// TIA Portal project "ConveyorBeltSystem" (V15)
// The purpose of project is to create a transport string system

(* hardware
DEVICE "S7-1200 station_1"  S7-1200 Station
   slot 0: "Rack_0"  S7-1200 Rack  Rack  V1.0
   slot 1: "PLC_1"  CPU 1214C DC/DC/DC  6ES7 214-1AG40-0XB0  V4.2
*)

// ===== PLC "PLC_1"  CPU 1214C DC/DC/DC =====

VAR_GLOBAL   // PLC tag table "Default tag table"
   "Takeoff_at_End3" AT %I0.5 : Bool;
   "Regulation" AT %I0.6 : Bool;   // ustawienie trybu pracy: szybki / wolny
   "Divisor" AT %M1.0 : Bool;   // przelacznik
   "Divisor_Memory" AT %M1.1 : Bool;   // pamiec przelacznika
   "Conveyor_Belt_1_Input" AT %I0.1 : Bool;   // wejscie na transporter #1
   "Conveyor_Belt_2_Input" AT %I0.2 : Bool;   // wejscie na transporter #2 / potwierdzenie odebrania paczki dla transportera #1
   "Conveyor_Belt_1_Output" AT %Q0.1 : Bool;   // wyjscie transporera #1 - sterowanie silnikiem
   "Conveyor_Belt_3_Input" AT %I0.3 : Bool;   // wejscie na transporter #3 / potwierdzenie odebrania paczki dla transportera #2
   "Conveyor_Belt_2_Output" AT %Q0.2 : Bool;   // wyjscie transporera #2 - sterowanie silnikiem
   "Conveyor_Belt_3_Confirm" AT %I0.4 : Bool;   // potwierdzenie odebrania paczki
   "Conveyor_Belt_3_Output" AT %Q0.3 : Bool;   // wyjscie transporera #3 - sterowanie silnikiem
   "Regulation_Edge" AT %M0.6 : Bool;   // zbocze regulacji trybow pracy
   "Conveyor_Belt_2_Status" AT %Q0.5 : Bool;   // sygnal wyjsciowy informujacy czy znajduje sie towar na koncu linii #2
   "Conveyor_Belt_3_Status" AT %Q0.6 : Bool;   // sygnal wyjsciowy informujacy czy znajduje sie towar na koncu linii #3
   "Conveyor_Belt_1_Status" AT %Q0.4 : Bool;   // sygnal wyjsciowy informujacy czy znajduje sie towar na koncu linii #1
   "Conveyor_Belt_1_Malfunction" AT %M500.0 : Bool;   // pamiec o wystapieniu awarii na transporterze #1
   "Conveyor_Belt_2_Malfunction" AT %M500.1 : Bool;   // pamiec o wystapieniu awarii na transporterze #2
   "Conveyor_Belt_3_Malfunction" AT %M500.2 : Bool;   // pamiec o wystapieniu awarii na transporterze #3
   "Tag_1" AT %M501.0 : Bool;
   "Tag_2" AT %M501.1 : Bool;
   "generator" AT %M30.0 : Bool;   // generator dla kanalow alarmowych
   "Conveyor_Belt_1_Alarm" AT %Q1.0 : Bool;   // wyjscie dla sygnalu awarii na transporterze #1
   "Conveyor_Belt_2_Alarm" AT %Q1.1 : Bool;   // wyjscie dla sygnalu awarii na transporterze #2
   "Conveyor_Belt_3_Alarm" AT %Q1.2 : Bool;   // wyjscie dla sygnalu awarii na transporterze #3
   "Emergency_Memory_1" AT %M500.3 : Bool;
   "Emergency_Memory_2" AT %M500.4 : Bool;
   "Emergency_Memory_3" AT %M500.5 : Bool;
   "Emergency_3_Confirm" AT %I1.2 : Bool;   // potwierdzenie awarii dla transportera #3
   "Emergency_2_Confirm" AT %I1.1 : Bool;   // potwierdzenie awarii dla transportera #2
   "Emergency_1_Confirm" AT %I1.0 : Bool;   // potwierdzenie awarii dla transportera #1
END_VAR

DATA_BLOCK "ConveyorBelt1_DB"   // DB1
{ S7_Optimized_Access := 'TRUE' }
VERSION : 0.1
// stored: InstanceOfName ConveyorBelt
"ConveyorBelt"
BEGIN
END_DATA_BLOCK

DATA_BLOCK "ConveyorBelt2_DB"   // DB2
{ S7_Optimized_Access := 'TRUE' }
VERSION : 0.1
// stored: InstanceOfName ConveyorBelt
"ConveyorBelt"
BEGIN
END_DATA_BLOCK

DATA_BLOCK "ConveyorBelt3_DB"   // DB3
{ S7_Optimized_Access := 'TRUE' }
VERSION : 0.1
// stored: InstanceOfName ConveyorBelt
"ConveyorBelt"
BEGIN
END_DATA_BLOCK

FUNCTION_BLOCK "ConveyorBelt"   // FB1, LAD
TITLE = Taśmociąg
{ S7_Optimized_Access := 'TRUE' }
VERSION : 0.1
// Blok funkcyjny odpowiedzialny za logikę pracy taśmociągu
   VAR_INPUT
      On_Line : Bool;   // podanie towaru na wejscie transportera
      Deliver_Confirm : Bool;   // potwierdzenie odbioru przez nastepna linie
      Malfunction_Confirm : Bool;   // potwierdzenie awarii przez operatora
   END_VAR
   VAR_OUTPUT
      Motor_Status : Bool;   // sygnal sterujacy silnikiem
      Malfunction : Bool;   // sygnal informujacy o awarii
      Output_Signal : Bool;   // sygnal informujacy, ze na koncu linii znajduje sie paczka
   END_VAR
   VAR
      Motor_Work : Bool;   // sygnal wyjsciowy informujacy o ladunku na koncu toru
      Blocked : Bool;   // sygnal ustawiajacy blokade transportera
      Photodiode_at_Start : Bool;   // status fotodiody umieszczonej na poczatku
      Counter_at_Start : Word;   // licznik towaru na wejsciu
      Photodiode_at_End : Bool;   // status fotodiody umieszczonej na koncu toru
      Counter_at_End : Word;   // licznik towaru na wyjsciu
      Work_Time : Time;   // czas pracy transportera
      IEC_Timer_0_Instance_2 : TP_TIME;
   END_VAR
   VAR RETAIN
      Package_Counter__Instance : CTUD_INT;
      Package_at_End_Counter_0_DB : CTU_INT;
   END_VAR
   VAR
      Photodiode_at_Start_Instance : "Photodiode";
      Photodiode_at_End_Instance : "Photodiode";
   END_VAR
   VAR RETAIN
      Counter_at_Start_Instance : CTU_INT;
   END_VAR
   VAR_TEMP
      Edge_Counter_at_Start_ : Bool;   // pamiec zbocza licznika na poczatku
      Edge_Counter_at_End : Bool;   // pamiec zbocza licznika na koncu
      Photodiode_End_Edge : Bool;   // pamiec zbocza fotodiody na koncu
      Photodiode_Start_Edge : Bool;   // pamiec zbocza fotodiody na poczatku
   END_VAR
   VAR_TEMP   // added for the SCL form of the ladder/FBD networks
      _w1 : Bool;
   END_VAR
BEGIN

REGION Network 1: Fotodioda 1: wykrycie towaru na początku
   // jesli nie ma blokady i fotodioda wykryje paczke ustaw jej sygnal
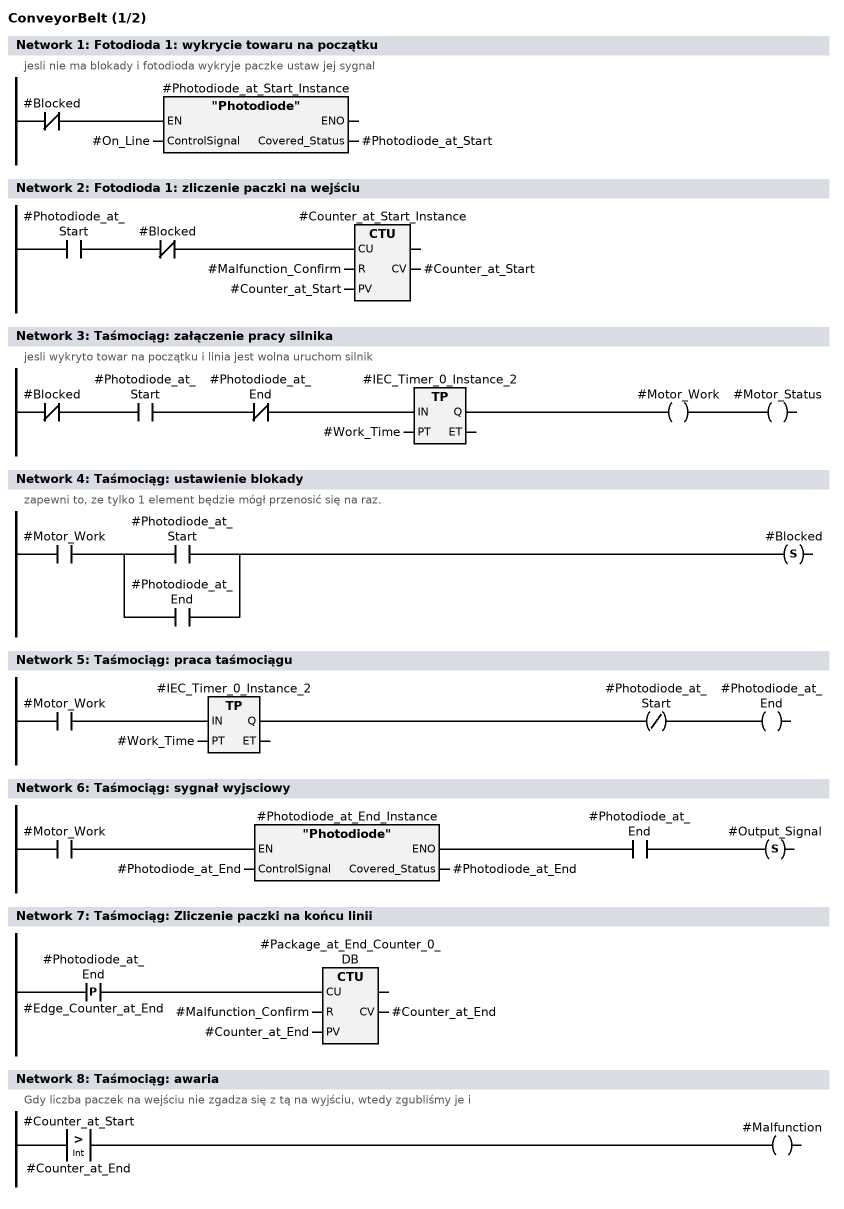
   RUNG wire#powerrail
      I_Contact( #Blocked )
      #Photodiode_at_Start_Instance(ControlSignal := #On_Line, Covered_Status => #Photodiode_at_Start)
   END_RUNG
   // the same network as SCL:
   IF NOT #Blocked THEN
       #Photodiode_at_Start_Instance(ControlSignal := #On_Line, Covered_Status => #Photodiode_at_Start);   // "Photodiode"
   END_IF;
END_REGION

REGION Network 2: Fotodioda 1: zliczenie paczki na wejściu
   #Counter_at_Start_Instance(CU := #Photodiode_at_Start AND NOT #Blocked,   // CTU
                           R := #Malfunction_Confirm,
                           PV := #Counter_at_Start,
                           CV => #Counter_at_Start);
END_REGION

REGION Network 3: Taśmociąg: załączenie pracy silnika
   // jesli wykryto towar na początku i linia jest wolna uruchom silnik
   #IEC_Timer_0_Instance_2(IN := NOT #Blocked AND #Photodiode_at_Start AND NOT #Photodiode_at_End,   // TP
                           PT := #Work_Time);
   #Motor_Work := #IEC_Timer_0_Instance_2.Q;
   #Motor_Status := #IEC_Timer_0_Instance_2.Q;
END_REGION

REGION Network 4: Taśmociąg: ustawienie blokady
   // zapewni to, ze tylko 1 element będzie mógł przenosić się na raz.
   RUNG wire#powerrail
      Contact( #Motor_Work )
      wire#w1
      Contact( #Photodiode_at_Start )
      wire#w2
      S_Coil( #Blocked )
   END_RUNG
   RUNG wire#w1
      Contact( #Photodiode_at_End )
   END_RUNG wire#w2
   // the same network as SCL:
   IF #Motor_Work AND (#Photodiode_at_Start OR #Photodiode_at_End) THEN #Blocked := TRUE; END_IF;
END_REGION

REGION Network 5: Taśmociąg: praca taśmociągu
   #IEC_Timer_0_Instance_2(IN := #Motor_Work, PT := #Work_Time);   // TP
   #Photodiode_at_Start := NOT #IEC_Timer_0_Instance_2.Q;
   #Photodiode_at_End := #IEC_Timer_0_Instance_2.Q;
END_REGION

REGION Network 6: Taśmociąg: sygnał wyjsciowy
   RUNG wire#powerrail
      Contact( #Motor_Work )
      #Photodiode_at_End_Instance(ControlSignal := #Photodiode_at_End, Covered_Status => #Photodiode_at_End)
      Contact( #Photodiode_at_End )
      S_Coil( #Output_Signal )
   END_RUNG
   // the same network as SCL:
   #Photodiode_at_End_Instance(EN := #Motor_Work,   // "Photodiode"
                           ControlSignal := #Photodiode_at_End,
                           Covered_Status => #Photodiode_at_End,
                           ENO => #_w1);
   IF #_w1 AND #Photodiode_at_End THEN #Output_Signal := TRUE; END_IF;
END_REGION

REGION Network 7: Taśmociąg: Zliczenie paczki na końcu linii
   #_w1 := #Photodiode_at_End AND NOT #Edge_Counter_at_End;   // rising edge of #Photodiode_at_End
   #Edge_Counter_at_End := #Photodiode_at_End;
   #Package_at_End_Counter_0_DB(CU := #_w1,   // CTU
                           R := #Malfunction_Confirm,
                           PV := #Counter_at_End,
                           CV => #Counter_at_End);
END_REGION

REGION Network 8: Taśmociąg: awaria
   // Gdy liczba paczek na wejściu nie zgadza się z tą na wyjściu, wtedy zgubliśmy je i
   RUNG wire#powerrail
      { S7_Templates := "SrcType := Int" } GT_Contact(in1 := #Counter_at_Start, in2 := #Counter_at_End)
      Coil( #Malfunction )
   END_RUNG
   // the same network as SCL:
   #Malfunction := #Counter_at_Start > #Counter_at_End;
END_REGION

REGION Network 9: Taśmociąg: potwiedzenie odbioru - reset linii
   // Następna linia podaje sygnał, że odebrała paczkę stąd też możemy zwolnić linię aby kolejna paczka mogła zostać przetransportowana
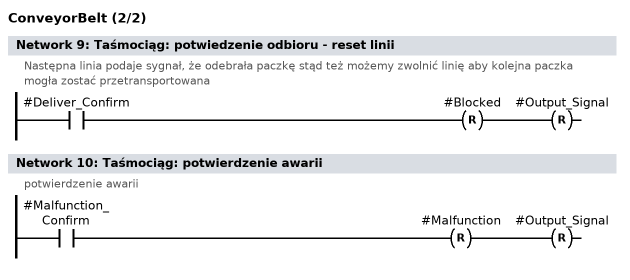
   RUNG wire#powerrail
      Contact( #Deliver_Confirm )
      R_Coil( #Blocked )
      R_Coil( #Output_Signal )
   END_RUNG
   // the same network as SCL:
   IF #Deliver_Confirm THEN
       #Blocked := FALSE;
       #Output_Signal := FALSE;
   END_IF;
END_REGION

REGION Network 10: Taśmociąg: potwierdzenie awarii
   // potwierdzenie awarii
   RUNG wire#powerrail
      Contact( #Malfunction_Confirm )
      R_Coil( #Malfunction )
      R_Coil( #Output_Signal )
   END_RUNG
   // the same network as SCL:
   IF #Malfunction_Confirm THEN
       #Malfunction := FALSE;
       #Output_Signal := FALSE;
   END_IF;
END_REGION
END_FUNCTION_BLOCK

FUNCTION_BLOCK "Photodiode"   // FB2, LAD
{ S7_Optimized_Access := 'TRUE' }
VERSION : 0.1
   VAR_INPUT
      ControlSignal : Bool;   // sygnal odebrany przez fotodiode
   END_VAR
   VAR_OUTPUT
      Covered_Status : Bool;   // sygnal stanu przysloniecia fotodiody
   END_VAR
   VAR
      IEC_Timer_0_Instance : TON_TIME;
   END_VAR
   VAR_TEMP
      edge : Bool;   // pamiec zbocza
   END_VAR
   VAR CONSTANT
      Cover_Delay : Time := T#450ms;   // czas opoznienia; zapobiega przypadkowemu zalaczeniu sie diody
   END_VAR
   VAR_TEMP   // added for the SCL form of the ladder/FBD networks
      _w1 : Bool;
   END_VAR
BEGIN

REGION Network 1: Fotodioda: wykrycie
   // Sygnał z fotodiody jest opóźniony aby zapobiec przed przypadkowym załączeniu się diody
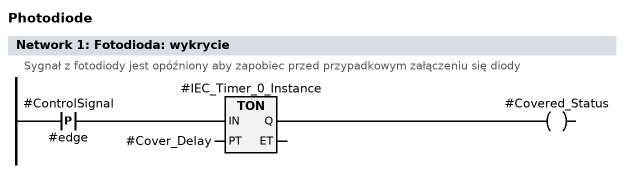
   #_w1 := #ControlSignal AND NOT #edge;   // rising edge of #ControlSignal
   #edge := #ControlSignal;
   #IEC_Timer_0_Instance(IN := #_w1, PT := #Cover_Delay);   // TON
   #Covered_Status := #IEC_Timer_0_Instance.Q;
END_REGION
END_FUNCTION_BLOCK

FUNCTION "EmergencyChannel" : Void   // FC1, LAD
{ S7_Optimized_Access := 'TRUE' }
VERSION : 0.1
   VAR_INPUT
      Pin_Generator : Bool;   // pamiec generatora szpilkowego
      Disruption : Bool;   // zakłócenie - sygnał o awarii
      Confirm : Bool;   // potwierdzenie reczne
   END_VAR
   VAR_OUTPUT
      Alarm : Bool;   // sygnalizacja awarii
   END_VAR
   VAR_IN_OUT
      Emergency_Memory : Bool;   // pamięć awarii
   END_VAR
   VAR_TEMP
      Emergency_Edge : Bool;   // pamięć zbocza awarii
      Generator_Edge_Memory : Bool;   // pamiec zbocza generatora
   END_VAR
   VAR_TEMP   // added for the SCL form of the ladder/FBD networks
      _w1 : Bool;
   END_VAR
BEGIN

REGION Network 1: Wykrycie awarii
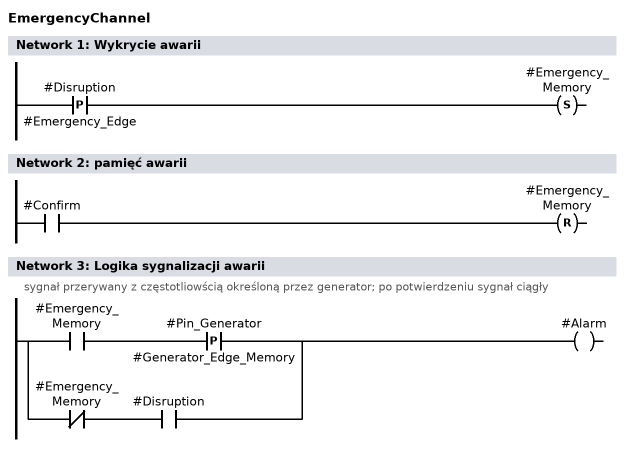
   RUNG wire#powerrail
      P_Contact(operand := #Disruption, bit := #Emergency_Edge)
      S_Coil( #Emergency_Memory )
   END_RUNG
   // the same network as SCL:
   #_w1 := #Disruption AND NOT #Emergency_Edge;   // rising edge of #Disruption
   #Emergency_Edge := #Disruption;
   IF #_w1 THEN #Emergency_Memory := TRUE; END_IF;
END_REGION

REGION Network 2: pamięć awarii
   RUNG wire#powerrail
      Contact( #Confirm )
      R_Coil( #Emergency_Memory )
   END_RUNG
   // the same network as SCL:
   IF #Confirm THEN #Emergency_Memory := FALSE; END_IF;
END_REGION

REGION Network 3: Logika sygnalizacji awarii
   // sygnał przerywany z częstotliowścią określoną przez generator; po potwierdzeniu sygnał ciągły
   RUNG wire#powerrail
      Contact( #Emergency_Memory )
      P_Contact(operand := #Pin_Generator, bit := #Generator_Edge_Memory)
      wire#w1
      Coil( #Alarm )
   END_RUNG
   RUNG wire#powerrail
      I_Contact( #Emergency_Memory )
      Contact( #Disruption )
   END_RUNG wire#w1
   // the same network as SCL:
   #_w1 := #Emergency_Memory AND #Pin_Generator AND NOT #Generator_Edge_Memory;   // rising edge of #Pin_Generator
   #Generator_Edge_Memory := #Pin_Generator;
   #Alarm := #_w1 OR (NOT #Emergency_Memory AND #Disruption);
END_REGION
END_FUNCTION

ORGANIZATION_BLOCK "Main"   // OB1, LAD, ProgramCycle
TITLE = "Main Program Sweep (Cycle)"
{ S7_Optimized_Access := 'TRUE' }
VERSION : 0.1
// Układ sekwencyjny 3 taśmociągów
   VAR_INPUT
      Initial_Call : Bool;   // Initial call of this OB
      Remanence : Bool;   // =True, if remanent data are available
   END_VAR
   VAR_TEMP   // added for the SCL form of the ladder/FBD networks
      _w1 : Bool;
   END_VAR
BEGIN

REGION Network 1: przełącznik binarny: ustawienie prędkości taśmociągu
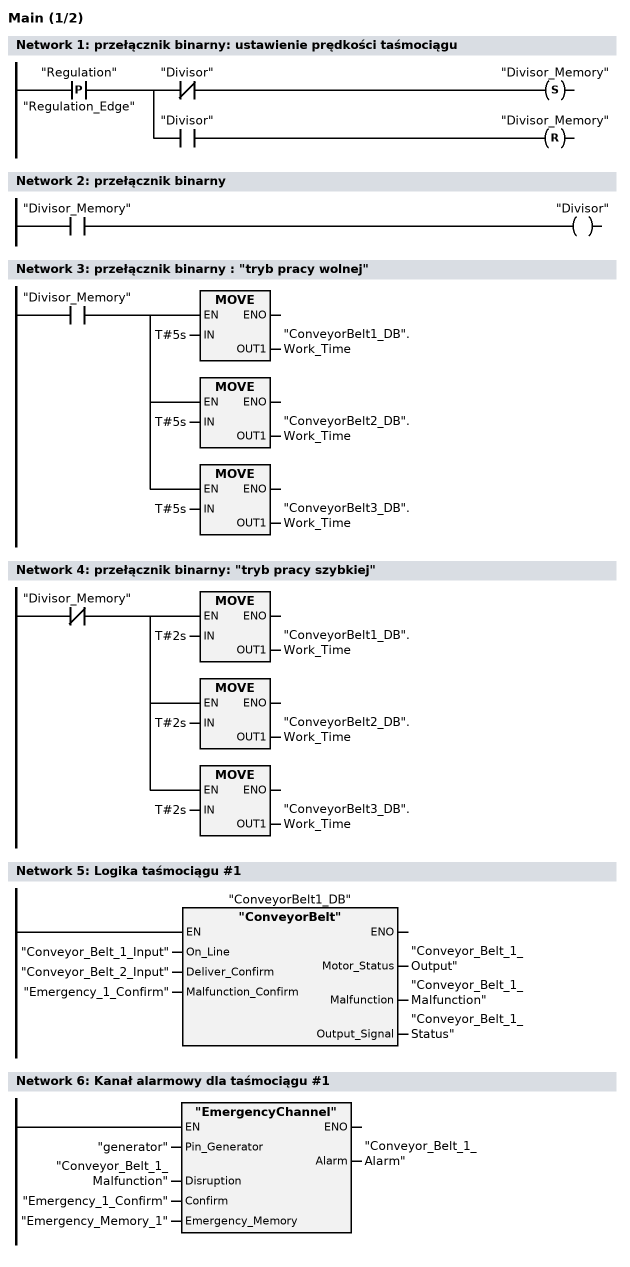
   RUNG wire#powerrail
      P_Contact(operand := "Regulation", bit := "Regulation_Edge")
      wire#w1
      I_Contact( "Divisor" )
      S_Coil( "Divisor_Memory" )
   END_RUNG
   RUNG wire#w1
      Contact( "Divisor" )
      R_Coil( "Divisor_Memory" )
   END_RUNG
   // the same network as SCL:
   #_w1 := "Regulation" AND NOT "Regulation_Edge";   // rising edge of "Regulation"
   "Regulation_Edge" := "Regulation";
   IF #_w1 AND NOT "Divisor" THEN "Divisor_Memory" := TRUE; END_IF;
   IF #_w1 AND "Divisor" THEN "Divisor_Memory" := FALSE; END_IF;
END_REGION

REGION Network 2: przełącznik binarny
   RUNG wire#powerrail
      Contact( "Divisor_Memory" )
      Coil( "Divisor" )
   END_RUNG
   // the same network as SCL:
   "Divisor" := "Divisor_Memory";
END_REGION

REGION Network 3: przełącznik binarny : "tryb pracy wolnej"
   RUNG wire#powerrail
      Contact( "Divisor_Memory" )
      wire#w1
      Move(in := T#5s, out1 => "ConveyorBelt1_DB".Work_Time)
   END_RUNG
   RUNG wire#w1
      Move(in := T#5s, out1 => "ConveyorBelt2_DB".Work_Time)
   END_RUNG
   RUNG wire#w1
      Move(in := T#5s, out1 => "ConveyorBelt3_DB".Work_Time)
   END_RUNG
   // the same network as SCL:
   IF "Divisor_Memory" THEN
       "ConveyorBelt1_DB".Work_Time := T#5s;
       "ConveyorBelt2_DB".Work_Time := T#5s;
       "ConveyorBelt3_DB".Work_Time := T#5s;
   END_IF;
END_REGION

REGION Network 4: przełącznik binarny: "tryb pracy szybkiej"
   RUNG wire#powerrail
      I_Contact( "Divisor_Memory" )
      wire#w1
      Move(in := T#2s, out1 => "ConveyorBelt1_DB".Work_Time)
   END_RUNG
   RUNG wire#w1
      Move(in := T#2s, out1 => "ConveyorBelt2_DB".Work_Time)
   END_RUNG
   RUNG wire#w1
      Move(in := T#2s, out1 => "ConveyorBelt3_DB".Work_Time)
   END_RUNG
   // the same network as SCL:
   IF NOT "Divisor_Memory" THEN
       "ConveyorBelt1_DB".Work_Time := T#2s;
       "ConveyorBelt2_DB".Work_Time := T#2s;
       "ConveyorBelt3_DB".Work_Time := T#2s;
   END_IF;
END_REGION

REGION Network 5: Logika taśmociągu #1
   RUNG wire#powerrail
      "ConveyorBelt1_DB"(On_Line := "Conveyor_Belt_1_Input", Deliver_Confirm := "Conveyor_Belt_2_Input", Malfunction_Confirm := "Emergency_1_Confirm", Motor_Status => "Conveyor_Belt_1_Output", Malfunction => "Conveyor_Belt_1_Malfunction", Output_Signal => "Conveyor_Belt_1_Status")
   END_RUNG
   // the same network as SCL:
   "ConveyorBelt1_DB"(On_Line := "Conveyor_Belt_1_Input",   // "ConveyorBelt"
                      Deliver_Confirm := "Conveyor_Belt_2_Input",
                      Malfunction_Confirm := "Emergency_1_Confirm",
                      Motor_Status => "Conveyor_Belt_1_Output",
                      Malfunction => "Conveyor_Belt_1_Malfunction",
                      Output_Signal => "Conveyor_Belt_1_Status");
END_REGION

REGION Network 6: Kanał alarmowy dla taśmociągu #1
   RUNG wire#powerrail
      "EmergencyChannel"(Pin_Generator := "generator", Disruption := "Conveyor_Belt_1_Malfunction", Confirm := "Emergency_1_Confirm", Emergency_Memory := "Emergency_Memory_1", Alarm => "Conveyor_Belt_1_Alarm")
   END_RUNG
   // the same network as SCL:
   "EmergencyChannel"(Pin_Generator := "generator",
                      Disruption := "Conveyor_Belt_1_Malfunction",
                      Confirm := "Emergency_1_Confirm",
                      Emergency_Memory := "Emergency_Memory_1",
                      Alarm => "Conveyor_Belt_1_Alarm");
END_REGION

REGION Network 7: Logika taśmociągu #2
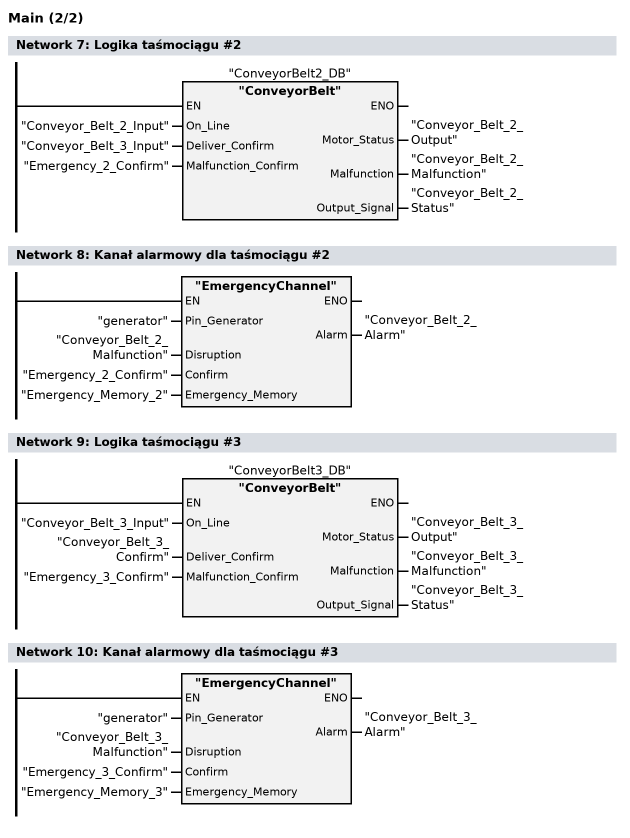
   RUNG wire#powerrail
      "ConveyorBelt2_DB"(On_Line := "Conveyor_Belt_2_Input", Deliver_Confirm := "Conveyor_Belt_3_Input", Malfunction_Confirm := "Emergency_2_Confirm", Motor_Status => "Conveyor_Belt_2_Output", Malfunction => "Conveyor_Belt_2_Malfunction", Output_Signal => "Conveyor_Belt_2_Status")
   END_RUNG
   // the same network as SCL:
   "ConveyorBelt2_DB"(On_Line := "Conveyor_Belt_2_Input",   // "ConveyorBelt"
                      Deliver_Confirm := "Conveyor_Belt_3_Input",
                      Malfunction_Confirm := "Emergency_2_Confirm",
                      Motor_Status => "Conveyor_Belt_2_Output",
                      Malfunction => "Conveyor_Belt_2_Malfunction",
                      Output_Signal => "Conveyor_Belt_2_Status");
END_REGION

REGION Network 8: Kanał alarmowy dla taśmociągu #2
   RUNG wire#powerrail
      "EmergencyChannel"(Pin_Generator := "generator", Disruption := "Conveyor_Belt_2_Malfunction", Confirm := "Emergency_2_Confirm", Emergency_Memory := "Emergency_Memory_2", Alarm => "Conveyor_Belt_2_Alarm")
   END_RUNG
   // the same network as SCL:
   "EmergencyChannel"(Pin_Generator := "generator",
                      Disruption := "Conveyor_Belt_2_Malfunction",
                      Confirm := "Emergency_2_Confirm",
                      Emergency_Memory := "Emergency_Memory_2",
                      Alarm => "Conveyor_Belt_2_Alarm");
END_REGION

REGION Network 9: Logika taśmociągu #3
   RUNG wire#powerrail
      "ConveyorBelt3_DB"(On_Line := "Conveyor_Belt_3_Input", Deliver_Confirm := "Conveyor_Belt_3_Confirm", Malfunction_Confirm := "Emergency_3_Confirm", Motor_Status => "Conveyor_Belt_3_Output", Malfunction => "Conveyor_Belt_3_Malfunction", Output_Signal => "Conveyor_Belt_3_Status")
   END_RUNG
   // the same network as SCL:
   "ConveyorBelt3_DB"(On_Line := "Conveyor_Belt_3_Input",   // "ConveyorBelt"
                      Deliver_Confirm := "Conveyor_Belt_3_Confirm",
                      Malfunction_Confirm := "Emergency_3_Confirm",
                      Motor_Status => "Conveyor_Belt_3_Output",
                      Malfunction => "Conveyor_Belt_3_Malfunction",
                      Output_Signal => "Conveyor_Belt_3_Status");
END_REGION

REGION Network 10: Kanał alarmowy dla taśmociągu #3
   RUNG wire#powerrail
      "EmergencyChannel"(Pin_Generator := "generator", Disruption := "Conveyor_Belt_3_Malfunction", Confirm := "Emergency_3_Confirm", Emergency_Memory := "Emergency_Memory_3", Alarm => "Conveyor_Belt_3_Alarm")
   END_RUNG
   // the same network as SCL:
   "EmergencyChannel"(Pin_Generator := "generator",
                      Disruption := "Conveyor_Belt_3_Malfunction",
                      Confirm := "Emergency_3_Confirm",
                      Emergency_Memory := "Emergency_Memory_3",
                      Alarm => "Conveyor_Belt_3_Alarm");
END_REGION
END_ORGANIZATION_BLOCK

ORGANIZATION_BLOCK "PinGenerator"   // OB30, LAD, CyclicInterrupt
{ S7_Optimized_Access := 'TRUE' }
VERSION : 0.1
   VAR_INPUT
      Initial_Call : Bool;   // Initial call of this OB
      Event_Count : Int;   // Events discarded
   END_VAR
BEGIN

REGION Network 1: Generator dla kanałów alarmowych taśmociągu
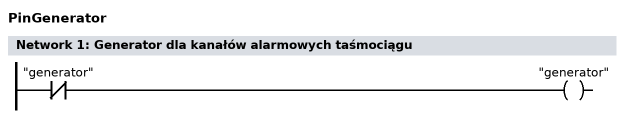
   RUNG wire#powerrail
      I_Contact( "generator" )
      Coil( "generator" )
   END_RUNG
   // the same network as SCL:
   "generator" := NOT "generator";
END_REGION
END_ORGANIZATION_BLOCK